FUNCTION_BLOCK TANK_MDL (* Tank Fill/Drain Model *)
  (* Standard: 61499-1 *)
  (* Version 0.5, 2004-09-04, JHC, Rockwell Automation, Made FEED, LEVEL REAL. *)
  (* Version 0.4, 2004-09-02, JHC, Rockwell Automation, Subclassed from E_CYCLE. *)
  (* Version 0.3, 2001-04-23, JHC, Rockwell Automation, Moved to fb.rt.process. *)
  (* Version 0.2, 2000-08-29, JHC, Rockwell Automation, Removed redundant "\n" *)
  (* Version 0.1, 2000-06-21, JHC, Rockwell Automation, Uses LibraryElement.dtd *)
  (* Version 0.0, 2000-04-28, JHC, Rockwell Automation *)
  (* Compiler header: package fb.rt.process; *)
  (* Compiler classdef: public class TANK_MDL extends E_CYCLE *)
  (* Compiler Java IBM VisualAge 3.0 *)
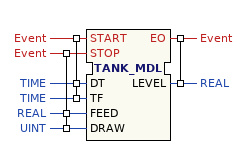
  EVENT_INPUT
    START WITH TF, DT; (* Start model *)
    STOP WITH FEED, DRAW; (* Stop model *)
  END_EVENT
  EVENT_OUTPUT
    EO WITH LEVEL; (* Level update *)
  END_EVENT
  VAR_INPUT
    DT : TIME := t#250ms; (* Simulation time interval *)
    TF : TIME := t#30s; (* Filling time at(FEED-DRAW)=100 *)
    FEED : REAL := 0; (* Liquid Feed Rate, 0-100%FS *)
    DRAW : UINT := 0; (* Liquid Drain Rate, 0-100%FS *)
  END_VAR
  VAR_OUTPUT
    LEVEL : REAL := 0; (* Liquid Level, 0-100%FS *)
  END_VAR
END_FUNCTION_BLOCK
